// TwinCAT 3 PLC project main
// ProgramVersion: 3.1.4024.0
// libraries:
//   Tc2_Standard, * (Beckhoff Automation GmbH)
//   Tc2_System, * (Beckhoff Automation GmbH)
//   Tc3_Module, * (Beckhoff Automation GmbH)
// project tree:
//   / GlobalTextList.TcGTLO, PlcTask.TcTTO, Visualization Manager.TcVMO (not stored)
//   POUs/ MAIN.TcPOU
//   VISUs/ Visu.TcVIS
// real-time tasks:
//   TASK PlcTask: cycle T#10ms, priority 20, ADS port 350

CONFIGURATION main
    RESOURCE PLC ON TwinCAT3
        TASK PlcTask(INTERVAL := T#10ms, PRIORITY := 20);
        PROGRAM MAIN WITH PlcTask : MAIN;
    END_RESOURCE
END_CONFIGURATION

// ---- POUs/MAIN.TcPOU
PROGRAM MAIN
VAR
	nPmeter AT %I* : REAL;
	nValue AT %Q* : BYTE;
END_VAR

//Lees de analoge waarde van de potentiometer op de PLC in en converteer naar een waarde van 0 tot en met 15 van het TYPE BYTE.
//Het kan zijn dat je de 'conversion operators' nodig hebt die je onder de 'input assistant' (F2-toets) terugvinden.

//Uitbreiding: Je kan nu de afzonderlijke bits van deze BYTE waarde toekennen aan de LED's op de PLC.
//Link vanuit de SW image de BYTE variable aan de afzonderlijke output values (type BOOL) door ‘All Types’ te selecteren (zie afbeelding hieronder).
//Vergeet natuurlijk geen offset mee te geven.
//Deze specifieert de bits van de BYTE variable die je wil koppelen met de corresponderende ouput van het type BOOL.
//Lees de analoge waarde van de potentiometer op de PLC in en converteer naar een waarde van 0 tot en met 15 van het type BYTE. 

nValue := REAL_TO_BYTE(nPmeter / 32767.0 * 15.0);

END_PROGRAM

// ---- VISUs/Visu.TcVIS
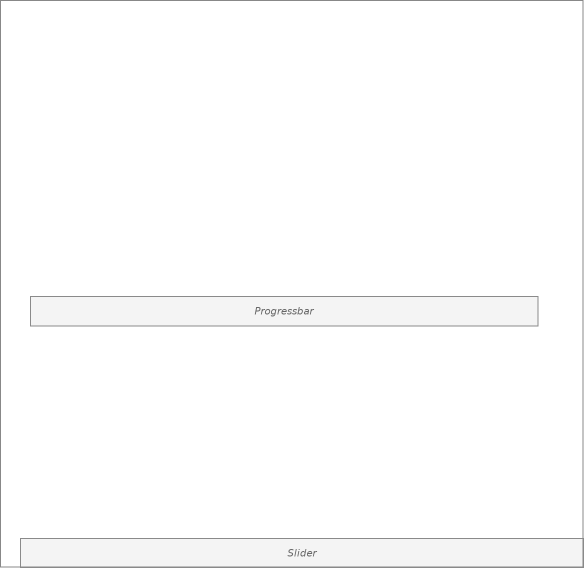
VISUALIZATION Visu  // 584x568
    Slider (20,538 564x30), variable: MAIN.nPmeter, scale 0..32767
    Progressbar (30,296 508x30), variable: MAIN.nValue
END_VISUALIZATION
